Fanuc KAREL source: kt00574.KL

-- PROVISIONAL review KL for V940-1; original PC SHA256 acc103fd47c4a1057b5f438588d2f2afaac701b8b5b9103e746cfb0c5f449f08
-- Incomplete behavior may be omitted. Consult companion uncertainty JSON. Do not deploy.
PROGRAM KT00574
%NOLOCKGROUP
VAR
  R1 : REAL
-- UNRESOLVED_DECL V2 type=000013
-- UNRESOLVED_DECL OUT type=000013
BEGIN
  -- V9_ZERO_TABLE_METADATA_HINT layout=0001; no indexed target words; source/name/runtime held
  -- UNRESOLVED_PC offsets 5-16; opcodes 2E,23
  -- UNRESOLVED_PC offsets 21-36; opcodes 2E,22,32,35
  -- UNRESOLVED_PC offsets 41-63; opcodes 21,49,90,4A
  -- UNRESOLVED_PC offsets 68-72; opcodes 7F
END KT00574
